FUNCTION_BLOCK FB_Maschinentuer
VAR_INPUT
	// Sensoreingang
	bDoorO	: BOOL;
	bDoorC	: BOOL;
	// Steuereingang
	bEnable	: BOOL;
	bOpen 	: BOOL;
	bClose 	: BOOL;
END_VAR
VAR_OUTPUT
	// Aktor Ausgang
	bVentil	: BOOL;
	// Zustände
	bError	: BOOL;
END_VAR
VAR
	nState : INT;
END_VAR

CASE nState OF
	0: // Tür geschlossen
	// Ausgänge setzen
	bVentil := TRUE;
	
	// Übergangsbedingung
	IF NOT bDoorC AND bEnable THEN
		nState := 3; // Tür schließen
	ELSIF bOpen THEN
		nState := 1; // Tür öffnen
	END_IF
	
	1: // Tür öffen
	// Ausgänge setzen
	bVentil := FALSE;
	
	// Übergangsbedingung
	IF NOT bDoorO THEN
		nState := nState + 1; // Tür geöffnet
	END_IF
	
	2: // Tür offen
	// Ausgänge setzen
	bVentil := FALSE;
	
	// Übergangsbedingung
	IF bClose AND bEnable THEN
		nState := nState + 1; // Tür schließen
	END_IF
	
	3: // Tür schließen
	// Ausgänge setzen
	bVentil := TRUE;
	
	// Übergangsbedingung
	IF NOT bDoorC THEN
		nState := 0; // Tür geöffnet
	END_IF
END_CASE

END_FUNCTION_BLOCK

(* stored: Version 1.1.0.1, ProductVersion 3.1.4024.15
   POU FB_Maschinentuer: Id {172d20d6-79a1-4c8e-b106-8cb5a964c781}, SpecialFunc None *)
